TYPE ST_DOS_Chanel_Diagnosis :
STRUCT
	bOvercurrent 		: BOOL;
	bOverload			: BOOL;
	bOpenLoad			: BOOL;
	bShortTo24V			: BOOL;
	PowersupplyMissing	: BOOL;
END_STRUCT
END_TYPE

(* stored: Version 1.1.0.1
   DUT ST_DOS_Chanel_Diagnosis: Id {84c712ae-7221-4653-b911-08ff2a499d7f} *)
